Staubli VAL3: RefreshList.pgx

program RefreshList()
  local num l_ni
begin
  //
  switch nPage
    //
    case 0
      if bListRefresh
        resize(sList,1,size(sFileList))
        for l_ni=0 to size(sFileList)-1
          sList[l_ni]=sFileList[l_ni]
        endFor
      endIf
    break
    //
    case 1
      if bListRefresh
        resize(sList,1,size(prd:pDemo))
        for l_ni=0 to size(prd:pDemo)-1
          sList[l_ni]="p"+toString("",l_ni+1)
        endFor
      endIf
    break
    case 2
    break
  endSwitch


end
